FUNCTION_BLOCK BFB_Reaction
  (* Standard: 61499-2 *)
  (* Version 0.1, 2016-00-31, hpea485, UOA *)
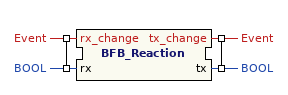
  EVENT_INPUT
    rx_change WITH rx;
  END_EVENT
  EVENT_OUTPUT
    tx_change WITH tx;
  END_EVENT
  VAR_INPUT
    rx : BOOL;
  END_VAR
  VAR_OUTPUT
    tx : BOOL;
  END_VAR
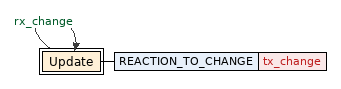
  EC_STATES
    Update : REACTION_TO_CHANGE -> tx_change;
  END_STATES
  EC_TRANSITIONS
    Update TO Update := rx_change;
  END_TRANSITIONS
  ALGORITHM REACTION_TO_CHANGE IN VHDL:
tx <= rx;
DONE <= '1';
  END_ALGORITHM
END_FUNCTION_BLOCK
